{attribute 'qualified_only'}
{attribute 'strict'}
TYPE eRunCondition :
(
	None := 0,
	SoC := 1,
	DischargeOverload := 2,
	BattFull := 3,
	ChargeOverload := 4,
	ManuallyStarted := 5,
	ManuallyStopped := 6
);
END_TYPE

(* stored: Version 1.1.0.1, ProductVersion 3.1.4026.18
   DUT eRunCondition: Id {037e5c7a-e232-49be-bcdc-e64005c97e9d} *)
